% RSLogix 500 project I2P Job 23 - Tyler_Vogt.RSS, saved by version 10.00.00.00 %
PROJECT "MLO2B"    % processor: Bul.1763 MicroLogix 1100 Series B %

PROGRAM FILES
  LAD 2   16 rungs

DATA FILES
  O0 OUTPUT  4 elements
  I1 INPUT  6 elements
  S2 STATUS  66 elements
  B3 BINARY  1 elements
  T4 TIMER  2 elements
  C5 COUNTER  2 elements
  R6 CONTROL  1 elements
  N7 INTEGER  1 elements
  F8 FLOAT  1 elements

LADDER 2
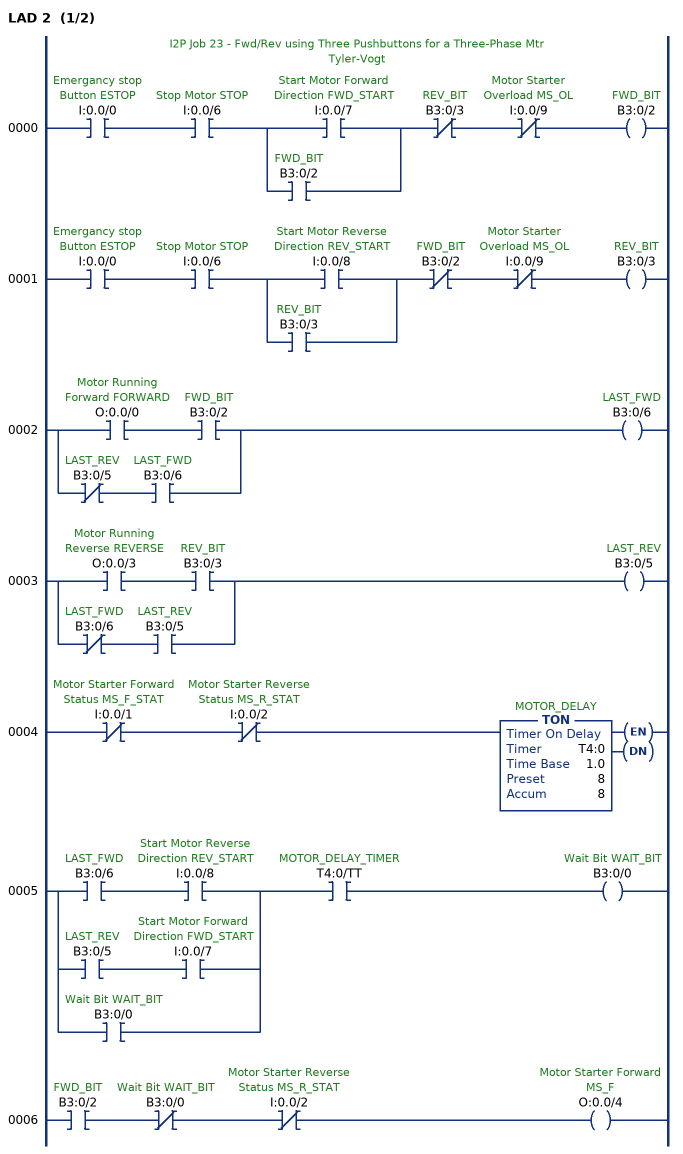
% Rung: 0 %  % edit flag set %
% I2P Job 23 - Fwd/Rev using Three Pushbuttons for a Three-Phase Mtr
% Tyler-Vogt %
SOR XIC I:0.0/0 XIC I:0.0/6 BST XIC I:0.0/7 NXB XIC B3:0/2 BND XIO B3:0/3 XIO I:0.0/9 OTE B3:0/2 EOR
%   I:0.0/0  ESTOP  "Emergancy stop Button" %
%   I:0.0/6  STOP  "Stop Motor" %
%   I:0.0/7  FWD_START  "Start Motor Forward Direction" %
%   B3:0/2  FWD_BIT %
%   B3:0/3  REV_BIT %
%   I:0.0/9  MS_OL  "Motor Starter Overload" %
% Rung: 1 %
SOR XIC I:0.0/0 XIC I:0.0/6 BST XIC I:0.0/8 NXB XIC B3:0/3 BND XIO B3:0/2 XIO I:0.0/9 OTE B3:0/3 EOR
%   I:0.0/0  ESTOP  "Emergancy stop Button" %
%   I:0.0/6  STOP  "Stop Motor" %
%   I:0.0/8  REV_START  "Start Motor Reverse Direction" %
%   B3:0/3  REV_BIT %
%   B3:0/2  FWD_BIT %
%   I:0.0/9  MS_OL  "Motor Starter Overload" %
% Rung: 2 %
SOR BST XIC O:0.0/0 XIC B3:0/2 NXB XIO B3:0/5 XIC B3:0/6 BND OTE B3:0/6 EOR
%   O:0.0/0  FORWARD  "Motor Running Forward" %
%   B3:0/2  FWD_BIT %
%   B3:0/5  LAST_REV %
%   B3:0/6  LAST_FWD %
% Rung: 3 %
SOR BST XIC O:0.0/3 XIC B3:0/3 NXB XIO B3:0/6 XIC B3:0/5 BND OTE B3:0/5 EOR
%   O:0.0/3  REVERSE  "Motor Running Reverse" %
%   B3:0/3  REV_BIT %
%   B3:0/6  LAST_FWD %
%   B3:0/5  LAST_REV %
% Rung: 4 %
SOR XIO I:0.0/1 XIO I:0.0/2 TON T4:0 1.0 8 8 EOR
%   I:0.0/1  MS_F_STAT  "Motor Starter Forward Status" %
%   I:0.0/2  MS_R_STAT  "Motor Starter Reverse Status" %
%   T4:0  MOTOR_DELAY %
% Rung: 5 %
SOR BST XIC B3:0/6 XIC I:0.0/8 NXB BST XIC B3:0/5 XIC I:0.0/7 NXB XIC B3:0/0 BND BND XIC T4:0/TT OTE B3:0/0 EOR
%   B3:0/6  LAST_FWD %
%   I:0.0/8  REV_START  "Start Motor Reverse Direction" %
%   B3:0/5  LAST_REV %
%   I:0.0/7  FWD_START  "Start Motor Forward Direction" %
%   B3:0/0  WAIT_BIT  "Wait Bit" %
%   T4:0/TT  MOTOR_DELAY_TIMER %
% Rung: 6 %
SOR XIC B3:0/2 XIO B3:0/0 XIO I:0.0/2 OTE O:0.0/4 EOR
%   B3:0/2  FWD_BIT %
%   B3:0/0  WAIT_BIT  "Wait Bit" %
%   I:0.0/2  MS_R_STAT  "Motor Starter Reverse Status" %
%   O:0.0/4  MS_F  "Motor Starter Forward" %

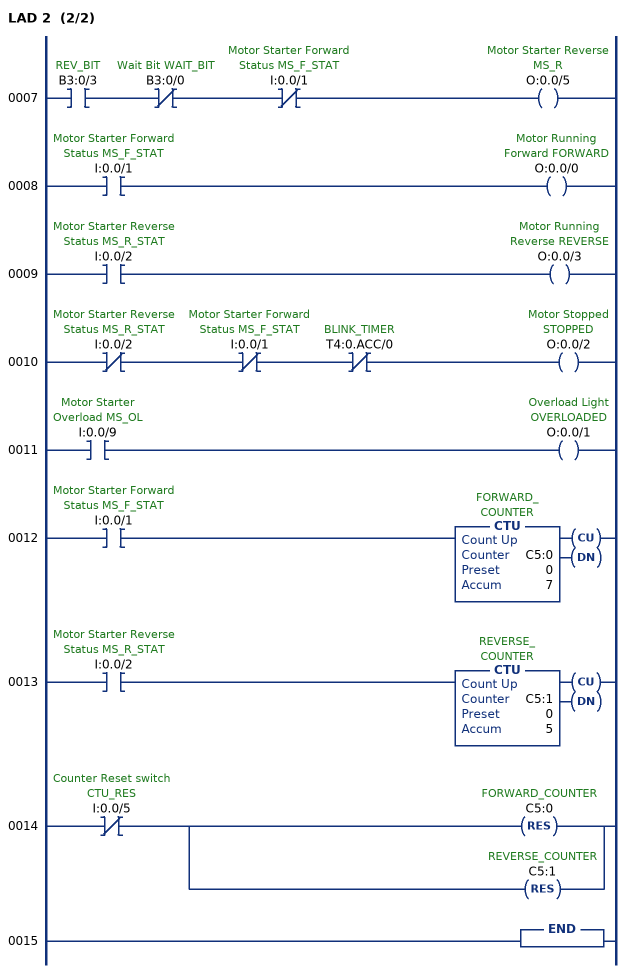
% Rung: 7 %
SOR XIC B3:0/3 XIO B3:0/0 XIO I:0.0/1 OTE O:0.0/5 EOR
%   B3:0/3  REV_BIT %
%   B3:0/0  WAIT_BIT  "Wait Bit" %
%   I:0.0/1  MS_F_STAT  "Motor Starter Forward Status" %
%   O:0.0/5  MS_R  "Motor Starter Reverse" %
% Rung: 8 %
SOR XIC I:0.0/1 OTE O:0.0/0 EOR
%   I:0.0/1  MS_F_STAT  "Motor Starter Forward Status" %
%   O:0.0/0  FORWARD  "Motor Running Forward" %
% Rung: 9 %
SOR XIC I:0.0/2 OTE O:0.0/3 EOR
%   I:0.0/2  MS_R_STAT  "Motor Starter Reverse Status" %
%   O:0.0/3  REVERSE  "Motor Running Reverse" %
% Rung: 10 %
SOR XIO I:0.0/2 XIO I:0.0/1 XIO T4:0.ACC/0 OTE O:0.0/2 EOR
%   I:0.0/2  MS_R_STAT  "Motor Starter Reverse Status" %
%   I:0.0/1  MS_F_STAT  "Motor Starter Forward Status" %
%   T4:0.ACC/0  BLINK_TIMER %
%   O:0.0/2  STOPPED  "Motor Stopped" %
% Rung: 11 %
SOR XIC I:0.0/9 OTE O:0.0/1 EOR
%   I:0.0/9  MS_OL  "Motor Starter Overload" %
%   O:0.0/1  OVERLOADED  "Overload Light" %
% Rung: 12 %
SOR XIC I:0.0/1 CTU C5:0 0 7 EOR
%   I:0.0/1  MS_F_STAT  "Motor Starter Forward Status" %
%   C5:0  FORWARD_COUNTER %
% Rung: 13 %
SOR XIC I:0.0/2 CTU C5:1 0 5 EOR
%   I:0.0/2  MS_R_STAT  "Motor Starter Reverse Status" %
%   C5:1  REVERSE_COUNTER %
% Rung: 14 %
SOR XIO I:0.0/5 BST RES C5:0 NXB RES C5:1 BND EOR
%   I:0.0/5  CTU_RES  "Counter Reset switch" %
%   C5:0  FORWARD_COUNTER %
%   C5:1  REVERSE_COUNTER %
% Rung: 15 %
SOR END EOR

OTHER DOCUMENTED ADDRESSES
  B3:0/1  ON_BIT  "On position bit"
  B3:0/4  YLW_LT_BIT
  B3:0/7  STOP_BIT  "Estop and Stop"
  FWD_JOG  "Forward Jog"
  I:0.0/3  AUTO_POS  "3 Position Selector Switch A Position"
  I:0.0/4  ON  "3 Position Selector Switch B Position"
  MOTOR  
  T4:0/DN  TIMER_DONE
  T4:0/EN  TIMER_ENABLED
  T4:1  FWD_DELAY

DATA TABLE (non-zero values as saved)
DATA B3
% B3:0 % 0X0040
DATA T4
% .PRE .ACC %
% T4:0 % 8 8
% T4:1 % 8 0
DATA C5
% .PRE .ACC %
% C5:0 % 0 7
% C5:1 % 0 5
